{attribute 'qualified_only'}
{attribute 'strict'}
TYPE Enum_ModuleEnableState :
(
	eDisabled				 := 0,
	eEnabled
);
END_TYPE

(* stored: Version 1.1.0.1, ProductVersion 3.1.4022.18
   DUT Enum_ModuleEnableState: Id {167df5f0-b717-44d2-9288-843d0eb0c45e} *)
